TYPE ST_GenComm_Params :
STRUCT
	IP					:	STRING	:=	'192.168.2.21';
	GenControlProtocol	: 	eGenControlProtocol := eGenControlProtocol.None;
END_STRUCT
END_TYPE

(* stored: Version 1.1.0.1, ProductVersion 3.1.4026.18
   DUT ST_GenComm_Params: Id {cc8c5794-9eff-42b9-832d-76db7b876d27} *)
